# EPICS substitutions: ek9000App/Db/EL2008_mbboDirect.substitutions
file EL2008.template
{       pattern
        {
                TERMINAL,

        }
        {
        }
}
